# EPICS autosave request: arucoUnwarpApp/Db/NDPluginArucoUnwarp_settings.req
$(P)$(R)MmPx
$(P)$(R)RefBoardSize
$(P)$(R)RefSquareSize
$(P)$(R)RefMarkerSize
$(P)$(R)RefBoardSquares
$(P)$(R)IncludeArUco
$(P)$(R)ArUcoDict
$(P)$(R)Scaling
file "NDPluginBase_settings.req", P=$(P), R=$(R)
